(* IEC 61131-3 sources: programs/VI-54/VI-54_20171205/VI-54_20171205/Stations/PLC_VI54/VI-54_171014/Class/_AlarmX1Para, 1 file *)

(* ---- _AlarmX1Para.st ---- *)
(*!
<Class
	Name               = "_AlarmX1Para"
	Revision           = "0.2"
	RealtimeTask       = "false"
	CyclicTask         = "false"
	BackgroundTask     = "false"
	Sigmatek           = "true"
	OSInterface        = "false"
	HighPriority       = "false"
	Automatic          = "false"
	UpdateMode         = "Prescan"
	SharedCommandTable = "true"
	Objectsize         = "(570,300)">
	<Channels>
		<Server
			Name           = "ClassSvr"
			Initialize     = "false"
			Visualized     = "true"
			WriteProtected = "false">
		</Server>
		<Client Name="Para1" Required="false" Internal="false"/>
	</Channels>
	<Network Name="_AlarmX1Para">
		<!-- List of Components in this network -->
		<Components>
			<Object
				Name       = "_base"
				Class      = "_AlarmX0Para"
				Position   = "(270,150)"
				Visualized = "true">
				<Channels>
					<Server Name="ClassSvr"/>
					<Client Name="Acknow"/>
					<Client Name="Config"/>
					<Client Name="Group"/>
				</Channels>
			</Object>
		</Components>
		<Comments>
		</Comments>
		<!-- List of Connections in this network -->
		<Connections>
			<Connection Source="this.ClassSvr" Destination="_base.ClassSvr" Vertices="(742,210),(570,240),"/>
			<Connection Source="_base.Config" Destination="this.Config" Vertices="(270,240),(38,210),"/>
			<Connection Source="_base.Acknow" Destination="this.Acknow" Vertices="(270,300),(38,270),"/>
			<Connection Source="_base.Group" Destination="this.Group" Vertices="(270,360),(38,330),"/>
		</Connections>
		<!-- Headerfiles -->
		<Options>
		</Options>
	</Network>
</Class>
*)
#pragma using _AlarmX0Para

_AlarmX1Para : CLASS
: _AlarmX0Para
  //Servers:
  //Clients:
	Para1 	: CltCh_DINT;
  //Variables:
  //Functions:

	FUNCTION VIRTUAL GLOBAL GetParaID
		VAR_INPUT
			ppara 	: ^UDINT;
		END_VAR
		VAR_OUTPUT
			retcode 	: UDINT;
		END_VAR;

	FUNCTION VIRTUAL GLOBAL GetParaVal
		VAR_INPUT
			ppara 	: ^DINT;
		END_VAR
		VAR_OUTPUT
			retcode 	: UDINT;
		END_VAR;
  //Tables:
	FUNCTION @STD
		VAR_OUTPUT
			ret_code	: CONFSTATES;
		END_VAR;
	FUNCTION GLOBAL TAB @CT_;
END_CLASS;

//*********************Inserted from .\_AlarmX1Para\_AlarmX1Para_00_00.st*********************

FUNCTION VIRTUAL GLOBAL _AlarmX1Para::GetParaID
  VAR_INPUT
    ppara		: ^UDINT;
  END_VAR
  VAR_OUTPUT
    retcode		: UDINT;
  END_VAR

  retcode := 1;

  if(IsClientConnected(#Para1) = TRUE) then
    ppara^ := (Para1.pCH)$UDINT;
  else
    ppara^ := 0;
  end_if;

END_FUNCTION
FUNCTION VIRTUAL GLOBAL _AlarmX1Para::GetParaVal
  VAR_INPUT
    ppara		: ^DINT;
  END_VAR
  VAR_OUTPUT
    retcode		: UDINT;
  END_VAR

  ppara^  := Para1.Read();
  retcode := 1;

END_FUNCTION
